// TIA Portal V18 export
FUNCTION_BLOCK "Z axis missing layer detection"   // FB3, LAD
TITLE = Description:
{ S7_Optimized_Access := 'TRUE' }
VERSION : 0.1
// Still in the development mode, not yet fully working.
// 
// Function block used to actively check if the positions of the Z1, Z2 axes are correct while printing. Missing layer detection is based on the check sum.
// stored: AutoNumber true, IsIECCheckEnabled false, IsRetainMemResEnabled false, MemoryReserve 100, SetENOAutomatically false, UDAEnableTagReadback false
   VAR_INPUT
      Mode : DInt;
      PrintStarted : Bool;
      PrintPaused : Bool;
      PrintEnded : Bool;
      Z1AxisPosition : DInt;
      Z1FeedStep : DInt;
      Z1Relative : Bool;
      Z2AxisPosition : DInt;
      Z2StepSize : DInt;
      Z2Relative : Bool;
      AmountOfLayers : DInt := 100;
      MotionMargin : DInt := 5;
      CompensationStepSize : DInt := 500;
      PrintingStepSize : DInt := 100;
   END_VAR
   VAR_OUTPUT
      Z1PredictedFinalPositionMinus : DInt;
      Z1PredictedFinalPosition : DInt;
      Z1PredictedFinalPositionPlus : DInt;
      Z2PredictedFinalPositionMinus : DInt;
      Z2PredictedFinalPosition : DInt;
      Z2PredictedFinalPositionPlus : DInt;
      MissingLayerStatus : Bool;   // 0 if the print is fine; 1 if the layer was skipped
      ErrorTime : Time;
   END_VAR
   VAR
      CheckSumStart : DInt;
      CheckSumMarginPlus : DInt;
      CheckSumMarginMinus : DInt;
      CheckSumActual : DInt;
      MachinePrintingInternal : Bool;
      MachinePrintingInternalM1 : Bool;
      Z1StartPosition : DInt;
      Z2StartPosition : DInt;
      Z1AddedDistanceInternal : DInt;
      Z2AddedDistanceInternal : DInt;
   END_VAR
   VAR_TEMP   // added for the SCL form of the ladder/FBD networks
      _w1 : Bool;
   END_VAR
BEGIN

REGION Network 1: Machine Printing Status
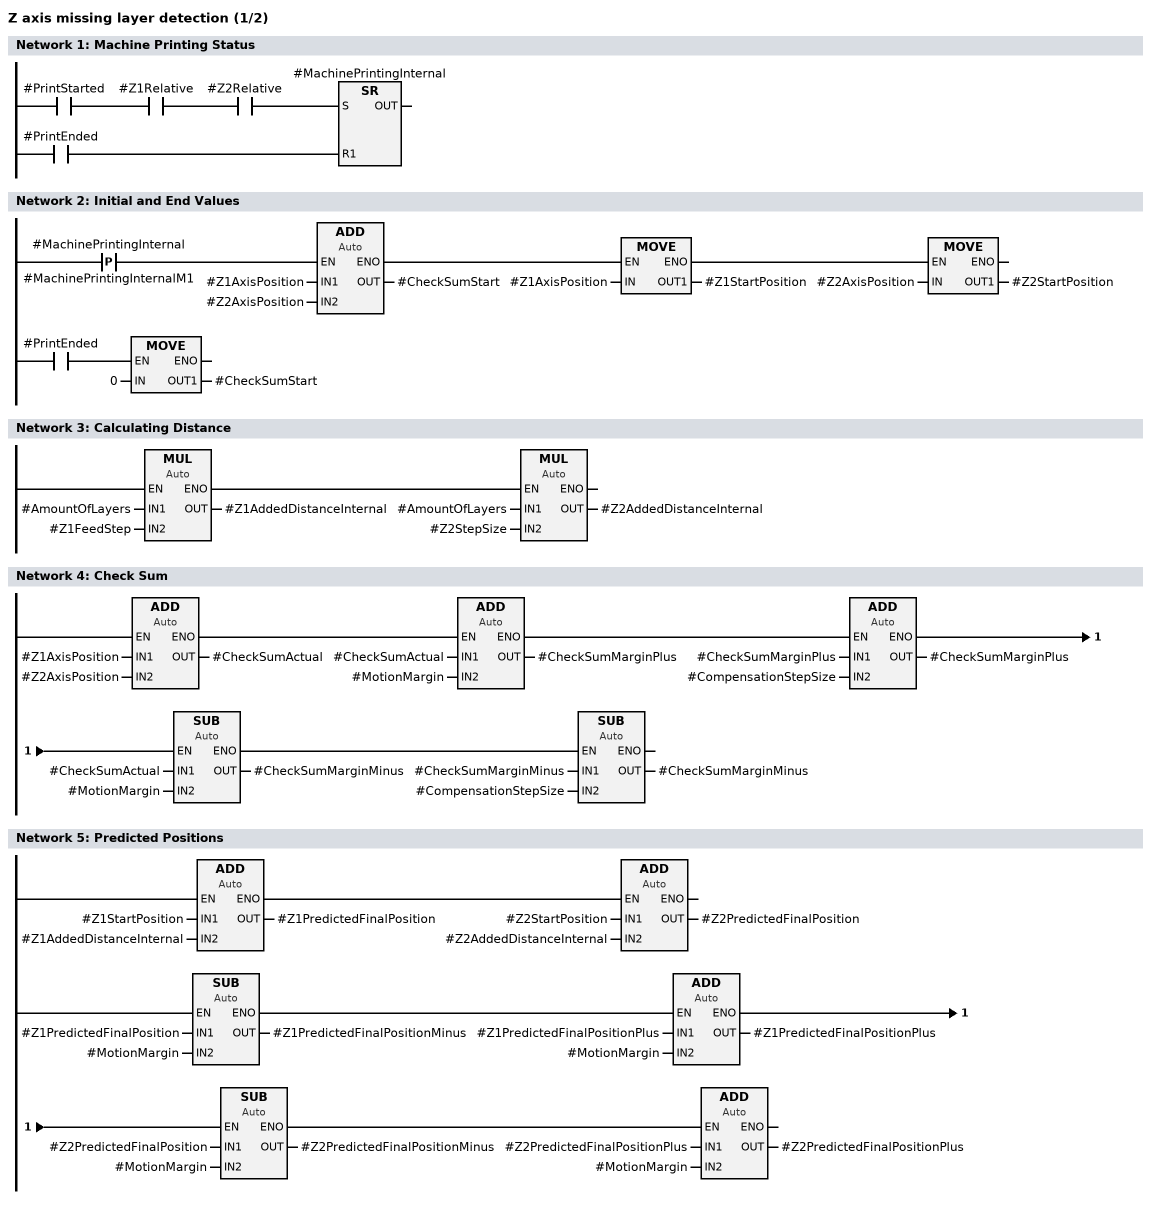
   RUNG wire#powerrail
      Contact( #PrintStarted )
      Contact( #Z1Relative )
      Contact( #Z2Relative )
      S_SR(operand := #MachinePrintingInternal, r1 := wire#w1)
   END_RUNG
   RUNG wire#powerrail
      Contact( #PrintEnded )
   END_RUNG wire#w1
   // the same network as SCL:
   IF #PrintStarted AND #Z1Relative AND #Z2Relative THEN
       #MachinePrintingInternal := TRUE;   // SR flip-flop
   END_IF;
   IF #PrintEnded THEN #MachinePrintingInternal := FALSE; END_IF;
END_REGION

REGION Network 2: Initial and End Values
   RUNG wire#powerrail
      P_Contact(operand := #MachinePrintingInternal, bit := #MachinePrintingInternalM1)
      Add(in1 := #Z1AxisPosition, in2 := #Z2AxisPosition, out => #CheckSumStart)
      Move(in := #Z1AxisPosition, out1 => #Z1StartPosition)
      Move(in := #Z2AxisPosition, out1 => #Z2StartPosition)
   END_RUNG
   RUNG wire#powerrail
      Contact( #PrintEnded )
      Move(in := 0, out1 => #CheckSumStart)
   END_RUNG
   // the same network as SCL:
   #_w1 := #MachinePrintingInternal AND NOT #MachinePrintingInternalM1;   // rising edge of #MachinePrintingInternal
   #MachinePrintingInternalM1 := #MachinePrintingInternal;
   IF #_w1 THEN
       #CheckSumStart := #Z1AxisPosition + #Z2AxisPosition;
       #Z1StartPosition := #Z1AxisPosition;
       #Z2StartPosition := #Z2AxisPosition;
   END_IF;
   IF #PrintEnded THEN #CheckSumStart := 0; END_IF;
END_REGION

REGION Network 3: Calculating Distance
   RUNG wire#powerrail
      Mul(in1 := #AmountOfLayers, in2 := #Z1FeedStep, out => #Z1AddedDistanceInternal)
      Mul(in1 := #AmountOfLayers, in2 := #Z2StepSize, out => #Z2AddedDistanceInternal)
   END_RUNG
   // the same network as SCL:
   #Z1AddedDistanceInternal := #AmountOfLayers * #Z1FeedStep;
   #Z2AddedDistanceInternal := #AmountOfLayers * #Z2StepSize;
END_REGION

REGION Network 4: Check Sum
   RUNG wire#powerrail
      Add(in1 := #Z1AxisPosition, in2 := #Z2AxisPosition, out => #CheckSumActual)
      Add(in1 := #CheckSumActual, in2 := #MotionMargin, out => #CheckSumMarginPlus)
      Add(in1 := #CheckSumMarginPlus, in2 := #CompensationStepSize, out => #CheckSumMarginPlus)
      Sub(in1 := #CheckSumActual, in2 := #MotionMargin, out => #CheckSumMarginMinus)
      Sub(in1 := #CheckSumMarginMinus, in2 := #CompensationStepSize, out => #CheckSumMarginMinus)
   END_RUNG
   // the same network as SCL:
   #CheckSumActual := #Z1AxisPosition + #Z2AxisPosition;
   #CheckSumMarginPlus := #CheckSumActual + #MotionMargin;
   #CheckSumMarginPlus := #CheckSumMarginPlus + #CompensationStepSize;
   #CheckSumMarginMinus := #CheckSumActual - #MotionMargin;
   #CheckSumMarginMinus := #CheckSumMarginMinus - #CompensationStepSize;
END_REGION

REGION Network 5: Predicted Positions
   RUNG wire#powerrail
      Add(in1 := #Z1StartPosition, in2 := #Z1AddedDistanceInternal, out => #Z1PredictedFinalPosition)
      Add(in1 := #Z2StartPosition, in2 := #Z2AddedDistanceInternal, out => #Z2PredictedFinalPosition)
   END_RUNG
   RUNG wire#powerrail
      Sub(in1 := #Z1PredictedFinalPosition, in2 := #MotionMargin, out => #Z1PredictedFinalPositionMinus)
      Add(in1 := #Z1PredictedFinalPositionPlus, in2 := #MotionMargin, out => #Z1PredictedFinalPositionPlus)
      Sub(in1 := #Z2PredictedFinalPosition, in2 := #MotionMargin, out => #Z2PredictedFinalPositionMinus)
      Add(in1 := #Z2PredictedFinalPositionPlus, in2 := #MotionMargin, out => #Z2PredictedFinalPositionPlus)
   END_RUNG
   // the same network as SCL:
   #Z1PredictedFinalPosition := #Z1StartPosition + #Z1AddedDistanceInternal;
   #Z2PredictedFinalPosition := #Z2StartPosition + #Z2AddedDistanceInternal;
   #Z1PredictedFinalPositionMinus := #Z1PredictedFinalPosition - #MotionMargin;
   #Z1PredictedFinalPositionPlus := #Z1PredictedFinalPositionPlus + #MotionMargin;
   #Z2PredictedFinalPositionMinus := #Z2PredictedFinalPosition - #MotionMargin;
   #Z2PredictedFinalPositionPlus := #Z2PredictedFinalPositionPlus + #MotionMargin;
END_REGION

REGION Network 6: Status
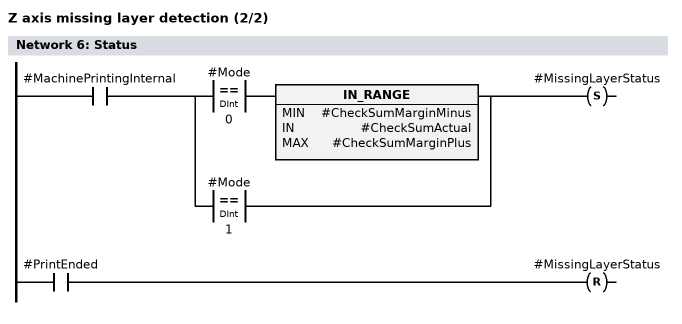
   RUNG wire#powerrail
      Contact( #MachinePrintingInternal )
      wire#w1
      { S7_Templates := "SrcType := DInt" } EQ_Contact(in1 := #Mode, in2 := 0)
      { S7_Templates := "SrcType := DInt" } InRange(min := #CheckSumMarginMinus, in := #CheckSumActual, max := #CheckSumMarginPlus)
      wire#w2
      S_Coil( #MissingLayerStatus )
   END_RUNG
   RUNG wire#w1
      { S7_Templates := "SrcType := DInt" } EQ_Contact(in1 := #Mode, in2 := 1)
   END_RUNG wire#w2
   RUNG wire#powerrail
      Contact( #PrintEnded )
      R_Coil( #MissingLayerStatus )
   END_RUNG
   // the same network as SCL:
   IF #MachinePrintingInternal AND (((#Mode = 0) AND (#CheckSumMarginMinus <= #CheckSumActual) AND (#CheckSumActual <= #CheckSumMarginPlus)) OR (#Mode = 1)) THEN
       #MissingLayerStatus := TRUE;
   END_IF;
   IF #PrintEnded THEN #MissingLayerStatus := FALSE; END_IF;
END_REGION
END_FUNCTION_BLOCK
